PROGRAM UserMode
VAR

(*GapMode*)
	UserGapPositionNew:LREAL:=20;//target
	UserGapVelocityNew:LREAL:=1;//target
	UserGapPositionDisplay:LREAL;//current
	UserGapVelocityDisplay:LREAL;//current
	//
	(**)
	btn_UserGapMove:BOOL;
	btn_UserGapStop:BOOL;
	(*Var*)
	fb_ton1:TON;
	fb_ton2:TON;
	fb_ton3:TON;
	(*Status*)
	State:DINT;
	Busy:BOOL;
	InitPowerDone:BOOL;
	InitCompensationDatasDone:BOOL;
	(*FB*)
	m_state: DINT;
	n_state: DINT;
	s_state: DINT;
	(*¼ì²âµ½ÏÞÎ»£¬»Ö¸´Move×´Ì¬*)
	FTrig_ReachLS: F_TRIG;
	FTrig_btn_GapMove: F_TRIG;
	GapOutRange: BOOL;
	(*PowerOff*)
	d_state: DINT;
	i: INT;
	j: INT;
	k: INT;
	moni_State:DINT;
	TargetPosLessThanCurrentPos:BOOL;
	PositiveMoving:BOOL;
	HysteresisMoving:BOOL;
	NoneHysteresisMoving:BOOL;
	(*Spectroscopy scanning Mode*)
	IsSSMotionMode:BOOL;
	RegularMotionMode:BOOL;
	SSMotionMode:BOOL;
	SS_StepSize:LREAL:=0.001;
	SS_StepNumber:INT:=10;
	SS_StepVelocity:LREAL:=1;
	SS_Move:BOOL;
	SS_Stop:BOOL;
	SS_MoveState:DINT;
	SS_StopState:DINT;
	SS_currentStep:DINT:=0;
	SS_StepSystemTime_Begin:ARRAY[0..100] OF ULINT;
	SS_StepSystemTime_End:ARRAY[0..100] OF ULINT;
	SS_StepCountTime:ARRAY[0..100] OF ULINT;
	SS_TimeCountBegin:BOOL;
	m: INT;
	SS_TON: TON;
	StepEachTime:TIME;
	StepEachTime_ms:INT:=1000;//ms
	SS_OTSTRUCT :OTSTRUCT ;
	SS_StartPositionDisplay:LREAL;
	RTRG_SS_StartPositionDisplay:R_TRIG;
	SS_InitStartPositionDone:BOOL;
	
	//
	min_SS_StepSize	: LREAL:=0;
	max_SS_StepSize	: LREAL:=200;
	inRange_SS_StepSize	: BOOL;
	//
	min_SS_StepNumber	: INT:=1;
	max_SS_StepNumber	: INT:=1000;
	inRange_SS_StepNumber	: BOOL;
	//
	min_SS_StepVelocity:LREAL:=0;
	max_SS_StepVelocity:LREAL:=1;
	inRange_SS_StepVelocity:BOOL;
	//
	min_StepEachTime_ms:INT:=100;
	max_StepEachTime_ms:INT:=10000;
	inRange_StepEachTime_ms:BOOL;
	l: INT;
	testa: BOOL;
	testb: BOOL;
	Threshold_GapChangeFlag: LREAL;
	Threshold_TaperChangeFlag: LREAL;
	TaperAndGapSafetyfactor: LREAL:=1;
	
		//
	//Global Chain protection-MPS
	Global_ChainProtection_MPS_StorageRingReady:BOOL;
	Global_ChainProtection_MPS_On: BOOL;
	Global_ChainProtection_MPS_MaxGapValue: LREAL;
	Global_ChainProtection_MPS_MoveVelocity: LREAL;
	Global_ChainProtection_MPS_Done: BOOL;
	//Global_ChainProtection_Error: BOOL;
	//Global_ChainProtection_ErrorID: INT;
	//Global_ChainProtection_ErrorDescription: STRING;
	Global_ChainProtection_MPS_ManualOperation:BOOL:=TRUE;
	Global_ChainProtection_MPS_FTRIG:F_TRIG;
	Global_ChainProtection_MPS_FTRIG_Manul:F_TRIG;
	Global_ChainProtection_MPS_TON:TON;
	Global_ChainProtection_MPS_Triggered:BOOL;
	Global_ChainProtection_MPS_In:BOOL;
	Global_ChainProtection_MPS_In1 AT%I* :BOOL;//下降沿表示触发
	Global_ChainProtection_MPS_In2 AT%I* :BOOL;
	Global_ChainProtection_MPS_State:DINT;
	Global_ChainProtection_MPS_Out1 AT%Q* :BOOL;//上升沿标识到达最大间隙，连锁保护成功
	Global_ChainProtection_MPS_Out2 AT%Q* :BOOL;
	Global_ChainProtection_MPS_TON_Stop2Move:TON;
	Global_ChainProtection_MPS_TON_Stop2Move_InTaperMode:TON;
	Global_ChainProtection_MPS_TON_Power2Move:TON;
	//Global Chain protection-EPS
	Global_ChainProtection_EPS_BeamLineReady:BOOL;
	Global_ChainProtection_EPS_On: BOOL;
	Global_ChainProtection_EPS_MaxGapValue: LREAL;
	Global_ChainProtection_EPS_MoveVelocity: LREAL;
	Global_ChainProtection_EPS_Done: BOOL;
	//Global_ChainProtection_Error: BOOL;
	//Global_ChainProtection_ErrorID: INT;
	//Global_ChainProtection_ErrorDescription: STRING;
	Global_ChainProtection_EPS_ManualOperation:BOOL:=TRUE;
	Global_ChainProtection_EPS_FTRIG:F_TRIG;
	Global_ChainProtection_EPS_FTRIG_Manul:F_TRIG;
	Global_ChainProtection_EPS_TON:TON;
	Global_ChainProtection_EPS_Triggered:BOOL;
	Global_ChainProtection_EPS_In:BOOL;
	Global_ChainProtection_EPS_In1 AT%I* :BOOL;//下降沿表示触发
	Global_ChainProtection_EPS_In2 AT%I* :BOOL;
	Global_ChainProtection_EPS_State:DINT;
	Global_ChainProtection_EPS_Out1 AT%Q* :BOOL;//上升沿标识到达最大间隙，连锁保护成功
	Global_ChainProtection_EPS_Out2 AT%Q* :BOOL;
	Global_ChainProtection_EPS_TON_Stop2Move:TON;
	Global_ChainProtection_EPS_TON_Stop2Move_InTaperMode:TON;
	Global_ChainProtection_EPS_TON_Power2Move:TON;
	//
	Threshold_motorsTargetPosCalculate:LREAL;
	
	PhaseShifterLinPositionNewTemp: LREAL;
		//OneKeyToMaxGap
	btn_OneKeyToMaxGap:BOOL;
	OneKeyToMaxGap_RTRIG:R_TRIG;
	OneKeyToMaxGap_TON:TON;
	OneKeyToMaxGap_Triggered:BOOL;
	OneKeyToMaxGap_State:DINT;
	OneKeyToMaxGap_TON_Stop2Move:TON;
	OneKeyToMaxGap_TON_Stop2Move_InTaperMode:TON;
	OneKeyToMaxGap_TON_Power2Move:TON;
	OneKeyToMaxGap_Done:BOOL;
END_VAR

IF NOT PositionBiasDone THEN
	RETURN;
END_IF
IF NOT loadParametersDone THEN
	RETURN;
END_IF
(*btn_Power On/Off*)
IF btn_Power AND NOT st_Power THEN
	btn_PowerOn:=TRUE;
	btn_Power:=FALSE;
END_IF
IF btn_Power AND st_Power THEN
	btn_PowerOff:=TRUE;
	btn_Power:=FALSE;
END_IF
IF btn_PowerOn THEN
	A_PowerOn();
END_IF
IF btn_PowerOff THEN
	A_PowerOff();
END_IF


(*补偿数据处理*)
A_InitCompensationData();

(*常规磁间隙开合*)
IF RegularMotionMode AND NOT SSMotionMode THEN
	A_RegularMotion();
END_IF

(*Spectroscopy scanning Mode*)
IF IsSSMotionMode THEN
	SSMotionMode:=TRUE;
	RegularMotionMode:=FALSE;
ELSE
	SSMotionMode:=FALSE;
	RegularMotionMode:=TRUE;
END_IF
IF	SSMotionMode AND NOT RegularMotionMode THEN
	A_SpectroscopyScanningMotion();
END_IF

A_CheckMotorsPos();

(*GlobalChainProtection*)
A_GlobalChainProtection_MPS();
A_GlobalChainProtection_EPS();

(*A_OneKeyToMaxGap*)
A_OneKeyToMaxGap();

ACTION A_CheckMotorsPos:
//
//目标位置速度超出阈值判断
//
//gap posiion
IF UserGapPositionNew<min_UserGapPositionNew OR UserGapPositionNew>max_UserGapPositionNew THEN
	inRange_UserGapPositionNew:=FALSE;
END_IF
IF UserGapPositionNew>=min_UserGapPositionNew AND UserGapPositionNew<=max_UserGapPositionNew THEN
	inRange_UserGapPositionNew:=TRUE;
END_IF
//gap velocity
IF UserGapVelocityNew<min_UserGapVelocityNew OR UserGapVelocityNew>max_UserGapVelocityNew THEN
	inRange_UserGapVelocityNew:=FALSE;
END_IF
IF UserGapVelocityNew>=min_UserGapVelocityNew AND UserGapVelocityNew<=max_UserGapVelocityNew THEN
	inRange_UserGapVelocityNew:=TRUE;
END_IF
//SS Mode
IF SS_StepSize<min_SS_StepSize OR SS_StepSize>max_SS_StepSize THEN
	inRange_SS_StepSize:=FALSE;
END_IF
IF SS_StepSize>=min_SS_StepSize AND SS_StepSize<=max_SS_StepSize THEN
	inRange_SS_StepSize:=TRUE;
END_IF
IF SS_StepNumber<min_SS_StepNumber OR SS_StepNumber>max_SS_StepNumber THEN
	inRange_SS_StepNumber:=FALSE;
END_IF
IF SS_StepNumber>=min_SS_StepNumber AND SS_StepNumber<=max_SS_StepNumber THEN
	inRange_SS_StepNumber:=TRUE;
END_IF
IF SS_StepVelocity<min_SS_StepVelocity OR SS_StepVelocity>max_SS_StepVelocity THEN
	inRange_SS_StepVelocity:=FALSE;
END_IF
IF SS_StepVelocity>=min_SS_StepVelocity AND SS_StepVelocity<=max_SS_StepVelocity THEN
	inRange_SS_StepVelocity:=TRUE;
END_IF
IF StepEachTime_ms<min_StepEachTime_ms OR StepEachTime_ms>max_StepEachTime_ms THEN
	inRange_StepEachTime_ms:=FALSE;
END_IF
IF StepEachTime_ms>=min_StepEachTime_ms AND StepEachTime_ms<=max_StepEachTime_ms THEN
	inRange_StepEachTime_ms:=TRUE;
END_IF


//
//输入速度和位置保护
//
IF btn_UserGapMove  AND NOT SSMotionMode AND RegularMotionMode THEN
	IF NOT inRange_UserGapPositionNew THEN
		btn_UserGapStop:=TRUE;
		btn_UserGapMove:=FALSE;
		Error:=TRUE;
		ErrorId:=801;
		ErrorDescription:='target Gap position out of range,please check';
		RETURN;
	ELSE
		//btn_UserGapStop:=FALSE;
		Error:=FALSE;
		ErrorId:=0;
		ErrorDescription:='';	
	END_IF
	IF NOT inRange_UserGapVelocityNew THEN
		btn_UserGapStop:=TRUE;
		btn_UserGapMove:=FALSE;
		Error:=TRUE;
		ErrorId:=802;
		ErrorDescription:='target Gap velocity out of range,please check';
		RETURN;
	ELSE
		//btn_UserGapStop:=FALSE;
		Error:=FALSE;
		ErrorId:=0;
		ErrorDescription:='';
	END_IF
END_IF

//
//运动过程中，监控目标位置速度
//
IF moveStatusPhaseShifterLin THEN
	IF NOT inRange_UserGapPositionNew THEN
		btn_UserGapStop:=TRUE;
		Error:=TRUE;
		ErrorId:=805;
		ErrorDescription:='target Gap position out of range in moving process!';
		FB_PlcEmergencyStop();
	END_IF
	IF NOT inRange_UserGapVelocityNew THEN
		btn_UserGapStop:=TRUE;
		Error:=TRUE;
		ErrorId:=806;
		ErrorDescription:='target Gap velocity out of range in moving process!';
		FB_PlcEmergencyStop();
	END_IF
END_IF
//
//运动过程中，监控每一个轴的目标位置，目标位置若超出阈值，Emergency
//
IF moveStatusPhaseShifterLin THEN
		IF PhaseShifterLinPositionNew<min_UserGapPositionNew OR PhaseShifterLinPositionNew>max_UserGapPositionNew THEN
			btn_UserGapStop:=TRUE;
			Error:=TRUE;
			ErrorId:=809;
			ErrorDescription:='target PhaseShifterLinPositionNew out of range in moving process!';
			FB_PlcEmergencyStop();
		END_IF
END_IF
END_ACTION

ACTION A_GlobalChainProtection_EPS:
//硬线输入定义
Global_ChainProtection_EPS_In:=Global_ChainProtection_EPS_In1 AND Global_ChainProtection_EPS_In2;
//硬线输出定义
Global_ChainProtection_EPS_Out1:=Global_ChainProtection_EPS_Done;
Global_ChainProtection_EPS_Out2:=Global_ChainProtection_EPS_Done;
//总开关
IF NOT Global_ChainProtection_EPS_On THEN
	RETURN;
END_IF
//判断插入件状态，是否就位
//IF NOT IDControlReady THEN
//	Global_ChainProtection_EPS_Done:=FALSE;
//	Error:= TRUE;
//	ErrorID:= 1501;
//	ErrorDescription:='ID NOT READY!';
//	RETURN;
//END_IF
//判断储存环是否给出就位信号，暂时由参数表给出TRUE，最终将由IOC接受PV
IF 	NOT Global_ChainProtection_EPS_BeamLineReady THEN
	Global_ChainProtection_EPS_Done:=FALSE;
	Error:= TRUE;
	ErrorID:= 1503;
	ErrorDescription:='Global_ChainProtection_EPS_BeamLineReady NOT Ready';
	RETURN;
END_IF
//
//全局连锁保护程序开始
//
//0.检测到下降沿，触发
//1.判断电机是否在开启状态,没有就打开电源
//2.判断是否在Moving状态,若有就Stop
//3.将磁间隙打开到至最大阈值
//4.到位后给出反馈，且安全PLC触发
Global_ChainProtection_EPS_FTRIG(CLK:=Global_ChainProtection_EPS_In);
IF Global_ChainProtection_EPS_FTRIG.Q THEN
	Global_ChainProtection_EPS_Triggered:=TRUE;
END_IF
Global_ChainProtection_EPS_FTRIG_Manul(CLK:=Global_ChainProtection_EPS_ManualOperation);
IF Global_ChainProtection_EPS_FTRIG_Manul.Q THEN
	Global_ChainProtection_EPS_Triggered:=TRUE;
END_IF
IF Global_ChainProtection_EPS_Triggered THEN
	CASE Global_ChainProtection_EPS_State OF
		0://1.判断电机是否在开启状态,没有就打开电源
			IF st_Power=1 THEN
				Global_ChainProtection_EPS_State:=1;
			ELSE
				btn_PowerOn:=TRUE;
				IF btn_PowerOn THEN
					A_PowerOn();
				END_IF
			END_IF
		1://1.判断是否在谱学扫描模式，如果是，则切换回正常运动模式
			IF IsSSMotionMode THEN
				SS_Stop:=TRUE;
				IsSSMotionMode:=FALSE;
			END_IF
			Global_ChainProtection_EPS_State:=2;
		2://判断是否在taper，如果在taper,则判断是否在运动，如果是，则停止运动,0.5sh后，转入下一步
			(*IF TaperOrNot THEN
				IF moveStatusLeftTop OR moveStatusRightTop OR moveStatusLeftBottom OR moveStatusRightBottom THEN
					btn_UserGapStop:=TRUE;
				ELSE
					Global_ChainProtection_EPS_TON_Stop2Move_InTaperMode(PT:=T#0.5S);
					Global_ChainProtection_EPS_TON_Stop2Move_InTaperMode.IN:=TRUE;
					IF Global_ChainProtection_EPS_TON_Stop2Move_InTaperMode.Q THEN
						TaperOrNot:=FALSE;//关闭taper模式
						Global_ChainProtection_EPS_State:=3;
					END_IF
				END_IF
			ELSE
			*)
				Global_ChainProtection_EPS_State:=3;
			//END_IF
		3://3.判断是否在Moving状态,若有就Stop.Taper模式已处理完，此处开始走正常GAP开合逻辑
			IF moveStatusPhaseShifterLin THEN
				btn_UserGapStop:=TRUE;
			ELSE
				Global_ChainProtection_EPS_TON_Stop2Move(PT:=T#0.5S);
				Global_ChainProtection_EPS_TON_Stop2Move.IN:=TRUE;
				IF Global_ChainProtection_EPS_TON_Stop2Move.Q THEN
					Global_ChainProtection_EPS_State:=4;
				END_IF
			END_IF
		4://当前磁间隙如何和最大磁间隙差别不大，不超过0.1，则直接保护
			IF ABS(UserGapPositionDisplay-Global_ChainProtection_EPS_MaxGapValue)<=0.1 THEN
				Global_ChainProtection_EPS_Done:=TRUE;
				Plc_EmergencyStop:=FALSE;	
				Error:=TRUE;
				ErrorID:=1506;
				ErrorDescription:='EPS Triggered,but ABS(UserGapPositionDisplay-Global_ChainProtection_EPS_MaxGapValue)<=0.1 ';	
			ELSE
				Global_ChainProtection_EPS_State:=5;
			END_IF
		5://5.将磁间隙打开到至最大阈值
			Global_ChainProtection_EPS_TON(PT:=INT_TO_TIME(LREAL_TO_INT(Global_ChainProtection_EPS_MaxGapValue/Global_ChainProtection_EPS_MoveVelocity+30))*1000);
			Global_ChainProtection_EPS_TON.IN:=TRUE;
			Global_ChainProtection_EPS_TON_Power2Move(PT:=T#0.1S);
			Global_ChainProtection_EPS_TON_Power2Move.IN:=TRUE;
			UserGapPositionNew:=Global_ChainProtection_EPS_MaxGapValue;
			UserGapVelocityNew:=Global_ChainProtection_EPS_MoveVelocity;
			btn_UserGapMove:=TRUE;
			IF Global_ChainProtection_EPS_TON_Power2Move.Q THEN
				IF FB_MOVE.BCGapDone THEN
					Global_ChainProtection_EPS_State:=88;
				END_IF
			END_IF
			IF Global_ChainProtection_EPS_TON.Q THEN//如果150s后，还没有运动到指定gap，则报错
				Global_ChainProtection_EPS_State:=-100;
			END_IF
		88://4.到位后给出反馈，且安全PLC触发
			Global_ChainProtection_EPS_Done:=TRUE;
			Plc_EmergencyStop:=FALSE;	
			Error:=TRUE;
			ErrorID:=1504;
			ErrorDescription:='Global_ChainProtection_EPS Triggered ';	
		-100:
			Global_ChainProtection_EPS_Done:=FALSE;
			Error:=TRUE;
			ErrorID:=1505;
			ErrorDescription:='NOT MOVING TO MAXGAP';
	END_CASE
END_IF
END_ACTION

ACTION A_GlobalChainProtection_MPS:
//硬线输入定义
Global_ChainProtection_MPS_In:=Global_ChainProtection_MPS_In1 AND Global_ChainProtection_MPS_In2;
//硬线输出定义
Global_ChainProtection_MPS_Out1:=Global_ChainProtection_MPS_Done;
Global_ChainProtection_MPS_Out2:=Global_ChainProtection_MPS_Done;
//总开关
IF NOT Global_ChainProtection_MPS_On THEN
	RETURN;
END_IF
//判断插入件状态，是否就位
//IF NOT IDControlReady THEN
//	Global_ChainProtection_MPS_Done:=FALSE;
//	Error:= TRUE;
//	ErrorID:= 1401;
//	ErrorDescription:='ID NOT READY!';
//	RETURN;
//END_IF
//判断储存环是否给出就位信号，暂时由参数表给出TRUE，最终将由IOC接受PV
IF 	NOT Global_ChainProtection_MPS_StorageRingReady THEN
	Global_ChainProtection_MPS_Done:=FALSE;
	Error:= TRUE;
	ErrorID:= 1403;
	ErrorDescription:='StorageRingChainProtection NOT Ready';
	RETURN;
END_IF
//
//全局连锁保护程序开始
//
//0.检测到下降沿，触发
//1.判断电机是否在开启状态,没有就打开电源
//2.判断是否在Moving状态,若有就Stop
//3.将磁间隙打开到至最大阈值
//4.到位后给出反馈，且安全PLC触发
Global_ChainProtection_MPS_FTRIG(CLK:=Global_ChainProtection_MPS_In);
IF Global_ChainProtection_MPS_FTRIG.Q THEN
	Global_ChainProtection_MPS_Triggered:=TRUE;
END_IF
Global_ChainProtection_MPS_FTRIG_Manul(CLK:=Global_ChainProtection_MPS_ManualOperation);
IF Global_ChainProtection_MPS_FTRIG_Manul.Q THEN
	Global_ChainProtection_MPS_Triggered:=TRUE;
END_IF
IF Global_ChainProtection_MPS_Triggered THEN
	CASE Global_ChainProtection_MPS_State OF
		0://1.判断电机是否在开启状态,没有就打开电源
			IF st_Power=1 THEN
				Global_ChainProtection_MPS_State:=1;
			ELSE
				btn_PowerOn:=TRUE;
				IF btn_PowerOn THEN
					A_PowerOn();
				END_IF
			END_IF
		1://1.判断是否在谱学扫描模式，如果是，则切换回正常运动模式
			IF IsSSMotionMode THEN
				SS_Stop:=TRUE;
				IsSSMotionMode:=FALSE;
			END_IF
			Global_ChainProtection_MPS_State:=2;
		2://判断是否在taper，如果在taper,则判断是否在运动，如果是，则停止运动,0.5sh后，转入下一步
			(*IF TaperOrNot THEN
				IF moveStatusLeftTop OR moveStatusRightTop OR moveStatusLeftBottom OR moveStatusRightBottom THEN
					btn_UserGapStop:=TRUE;
				ELSE
					Global_ChainProtection_MPS_TON_Stop2Move_InTaperMode(PT:=T#0.5S);
					Global_ChainProtection_MPS_TON_Stop2Move_InTaperMode.IN:=TRUE;
					IF Global_ChainProtection_MPS_TON_Stop2Move_InTaperMode.Q THEN
						TaperOrNot:=FALSE;//关闭taper模式
						Global_ChainProtection_MPS_State:=3;
					END_IF
				END_IF
			ELSE
			*)
				Global_ChainProtection_MPS_State:=3;
			//END_IF
		3://3.判断是否在Moving状态,若有就Stop.Taper模式已处理完，此处开始走正常GAP开合逻辑
			IF moveStatusPhaseShifterLin THEN
				btn_UserGapStop:=TRUE;
			ELSE
				Global_ChainProtection_MPS_TON_Stop2Move(PT:=T#0.5S);
				Global_ChainProtection_MPS_TON_Stop2Move.IN:=TRUE;
				IF Global_ChainProtection_MPS_TON_Stop2Move.Q THEN
					Global_ChainProtection_MPS_State:=4;
				END_IF
			END_IF
		4://当前磁间隙如何和最大磁间隙差别不大，不超过0.1，则直接保护
			IF ABS(UserGapPositionDisplay-Global_ChainProtection_MPS_MaxGapValue)<=0.1 THEN
				Global_ChainProtection_MPS_Done:=TRUE;
				Plc_EmergencyStop:=FALSE;	
				Error:=TRUE;
				ErrorID:=1406;
				ErrorDescription:='MPS Triggered,but ABS(UserGapPositionDisplay-Global_ChainProtection_MPS_MaxGapValue)<=0.1 ';	
			ELSE
				Global_ChainProtection_MPS_State:=5;
			END_IF
		5://5.将磁间隙打开到至最大阈值
			Global_ChainProtection_MPS_TON(PT:=INT_TO_TIME(LREAL_TO_INT(Global_ChainProtection_MPS_MaxGapValue/Global_ChainProtection_MPS_MoveVelocity+30))*1000);
			Global_ChainProtection_MPS_TON.IN:=TRUE;
			Global_ChainProtection_MPS_TON_Power2Move(PT:=T#0.1S);
			Global_ChainProtection_MPS_TON_Power2Move.IN:=TRUE;
			UserGapPositionNew:=Global_ChainProtection_MPS_MaxGapValue;
			UserGapVelocityNew:=Global_ChainProtection_MPS_MoveVelocity;
			btn_UserGapMove:=TRUE;
			IF Global_ChainProtection_MPS_TON_Power2Move.Q THEN
				IF FB_MOVE.BCGapDone THEN
					Global_ChainProtection_MPS_State:=88;
				END_IF
			END_IF
			IF Global_ChainProtection_MPS_TON.Q THEN//如果150s后，还没有运动到指定gap，则报错
				Global_ChainProtection_MPS_State:=-100;
			END_IF
		88://4.到位后给出反馈，且安全PLC触发
			Global_ChainProtection_MPS_Done:=TRUE;
			Plc_EmergencyStop:=FALSE;	
			Error:=TRUE;
			ErrorID:=1404;
			ErrorDescription:='Global_ChainProtection_MPS Triggered ';	
		-100:
			Global_ChainProtection_MPS_Done:=FALSE;
			Error:=TRUE;
			ErrorID:=1405;
			ErrorDescription:='NOT MOVING TO MAXGAP';
	END_CASE
END_IF
END_ACTION

ACTION A_InitCompensationData:
(*补偿开始*)
IF USE_SingleAxis_Compensation THEN
	//
	//1.目标位置解算
	//
	//左轴目标位置解算
	FOR	i:= 1 TO 17 DO
			IF UserGapPositionNew<M_Compensation[i+1].Gap AND UserGapPositionNew>=M_Compensation[i].Gap THEN
				IF i<>18 THEN
					PhaseShifterLinPositionNew:=(((UserGapPositionNew-M_Compensation[i].Gap)*(M_Compensation[i+1].PhaseShifterLin-M_Compensation[i].PhaseShifterLin))
							/(M_Compensation[i+1].Gap-M_Compensation[i].Gap))+M_Compensation[i].PhaseShifterLin;
					M_CompensationNumber:=i;
					InitCompensationDatasDone:=TRUE;
				ELSIF i=18 AND UserGapPositionNew=M_Compensation[i].Gap THEN		(*Gap=14µÄÌØÊâÇé¿ö*)
					(**)
					PhaseShifterLinPositionNew:=M_Compensation[i].PhaseShifterLin;
					M_CompensationNumber:=i;
					InitCompensationDatasDone:=TRUE;
				ELSE
					PhaseShifterLinPositionNew:=UserGapPositionNew;
					M_CompensationNumber:=i;
					InitCompensationDatasDone:=TRUE;
				END_IF
			END_IF
	END_FOR

	//显示位置反解算
	FOR k:= 1 TO 17 DO
			IF Pos_PhaseShifterLin<M_Compensation[k+1].PhaseShifterLin AND Pos_PhaseShifterLin>=M_Compensation[k].PhaseShifterLin THEN
				UserGapPositionDisplay:=((Pos_PhaseShifterLin-M_Compensation[k].PhaseShifterLin)*(M_Compensation[k+1].Gap-M_Compensation[k].Gap))
											/(M_Compensation[k+1].PhaseShifterLin-M_Compensation[k].PhaseShifterLin)+M_Compensation[k].Gap;
				UserGapPositionDisplay:=DINT_TO_LREAL(LREAL_TO_DINT(UserGapPositionDisplay*100000))/100000;
			END_IF
	END_FOR
END_IF
(*速度可以不用解算，直接用即可*)
PhaseShifterLinVelocityDisplay:=Velo_PhaseShifterLin;
//Gap velocity
UserGapVelocityDisplay:=DINT_TO_LREAL(LREAL_TO_DINT(PhaseShifterLinVelocityDisplay*100000))/100000;


(*解算单轴位置后，核验并做保护*)
IF ABS(PhaseShifterLinPositionNew-UserGapPositionNew)>Threshold_motorsTargetPosCalculate THEN
	ErrorID:=1601;
	Error:=TRUE;
	ErrorDescription:='Threshold_motorsTargetPosCalculate';
	FB_PlcEmergencyStop();
END_IF
END_ACTION

ACTION A_OneKeyToMaxGap:
//0.上升沿触发
//1.判断电机是否在开启状态,没有就打开电源
//2.判断是否在Moving状态,若有就Stop
//3.将磁间隙打开到至最大阈值
//4.到位后给出反馈
OneKeyToMaxGap_RTRIG(CLK:=btn_OneKeyToMaxGap);
IF OneKeyToMaxGap_RTRIG.Q THEN
	OneKeyToMaxGap_Triggered:=TRUE;
	OneKeyToMaxGap_Done:=FALSE;
END_IF
IF OneKeyToMaxGap_Triggered THEN
	CASE OneKeyToMaxGap_State OF
		0://1.判断电机是否在开启状态,没有就打开电源
			IF st_Power=1 THEN
				OneKeyToMaxGap_State:=1;
			ELSE
				btn_PowerOn:=TRUE;
				IF btn_PowerOn THEN
					A_PowerOn();
				END_IF
			END_IF
		1://1.判断是否在谱学扫描模式，如果是，则切换回正常运动模式
			IF IsSSMotionMode THEN
				SS_Stop:=TRUE;
				IsSSMotionMode:=FALSE;
			END_IF
			OneKeyToMaxGap_State:=2;
		2://判断是否在taper，如果在taper,则判断是否在运动，如果是，则停止运动,0.5sh后，转入下一步
			//IF TaperOrNot THEN
			//	IF moveStatusLeftTop OR moveStatusRightTop OR moveStatusLeftBottom OR moveStatusRightBottom THEN
			//		btn_UserGapStop:=TRUE;
			//	ELSE
			//		OneKeyToMaxGap_TON_Stop2Move_InTaperMode(PT:=T#0.5S);
			//		OneKeyToMaxGap_TON_Stop2Move_InTaperMode.IN:=TRUE;
			//		IF OneKeyToMaxGap_TON_Stop2Move_InTaperMode.Q THEN
			//			TaperOrNot:=FALSE;//关闭taper模式
			//			OneKeyToMaxGap_State:=3;
			//			OneKeyToMaxGap_TON_Stop2Move_InTaperMode.IN:=FALSE;
			//		END_IF
			//	END_IF
			//ELSE
				OneKeyToMaxGap_State:=3;
			//END_IF
		3://3.判断是否在Moving状态,若有就Stop.Taper模式已处理完，此处开始走正常GAP开合逻辑
			IF moveStatusPhaseShifterLin THEN
				btn_UserGapStop:=TRUE;
			ELSE
				OneKeyToMaxGap_TON_Stop2Move(PT:=T#0.5S);
				OneKeyToMaxGap_TON_Stop2Move.IN:=TRUE;
				IF OneKeyToMaxGap_TON_Stop2Move.Q THEN
					OneKeyToMaxGap_State:=4;
					OneKeyToMaxGap_TON_Stop2Move.IN:=FALSE;
				END_IF
			END_IF
		4://4.将磁间隙打开到至最大阈值
			OneKeyToMaxGap_TON(PT:=INT_TO_TIME(LREAL_TO_INT(max_UserGapPositionNew+30))*1000);
			OneKeyToMaxGap_TON.IN:=TRUE;
			OneKeyToMaxGap_TON_Power2Move(PT:=T#0.1S);
			OneKeyToMaxGap_TON_Power2Move.IN:=TRUE;
			UserGapPositionNew:=max_UserGapPositionNew;
			UserGapVelocityNew:=1;
			btn_UserGapMove:=TRUE;
			IF OneKeyToMaxGap_TON_Power2Move.Q THEN
				OneKeyToMaxGap_TON_Power2Move.IN:=FALSE;
				IF FB_MOVE.BCGapDone THEN
					OneKeyToMaxGap_State:=88;
				END_IF
			END_IF
			IF OneKeyToMaxGap_TON.Q THEN//如果150s后，还没有运动到指定gap，则报错
				OneKeyToMaxGap_TON.IN:=FALSE;
				OneKeyToMaxGap_State:=-100;
			END_IF
			IF  btn_UserGapStop THEN
				//
				OneKeyToMaxGap_State:=0;
				OneKeyToMaxGap_Triggered:=FALSE;
				btn_OneKeyToMaxGap:=FALSE;
				OneKeyToMaxGap_Triggered:=FALSE;
				OneKeyToMaxGap_State:=0;
			END_IF
		88://6.到位后给出反馈
			OneKeyToMaxGap_Done:=TRUE;	
			Error:=FALSE;
			ErrorID:=0;
			ErrorDescription:='';
			btn_OneKeyToMaxGap:=FALSE;
			OneKeyToMaxGap_Triggered:=FALSE;
			OneKeyToMaxGap_State:=0;
				
		-100:
			OneKeyToMaxGap_Done:=FALSE;
			Error:=TRUE;
			ErrorID:=1705;
			ErrorDescription:='OneKeyToMaxGap Fail';
			btn_OneKeyToMaxGap:=FALSE;
			OneKeyToMaxGap_Triggered:=FALSE;
			OneKeyToMaxGap_State:=0;
	END_CASE
END_IF
END_ACTION

ACTION A_PowerOff:
CASE d_state OF
		0:(*PowerOff*)
			FB_Power(Off:=TRUE);
				d_state:=1;
		1:
			IF NOT FB_power.OffStatus THEN
				d_state:=1;
			ELSE
				d_state:=88;
			END_IF
		88:(*ResetAllState*)
			btn_PowerOn:=FALSE;
			btn_UserGapMove:=FALSE;
			btn_UserGapStop:=FALSE;
			fb_ton1.IN:=FALSE;
			fb_ton2.IN:=FALSE;
			fb_ton3.IN:=FALSE;
			State:=0;
			Busy:=FALSE;
			InitPowerDone:=FALSE;
			InitCompensationDatasDone:=FALSE;
			Error:=FALSE;
			ErrorID:=0;
			m_state:=0;
			n_state:=0;
			s_state:=0;
			btn_PowerOff:=FALSE;
			d_state:=0;
			Led_Run:=FALSE;
			Led_Error:=FALSE;
			moni_State:=0;
			i:=0;
END_CASE
END_ACTION

ACTION A_PowerOn:
(****************************************************************
NAME:			A_PowerOn
DATA:			2018.1.9
VERSION:		1.0.0
DESCRIPTION:	
				ÉÏµãÃüÁîºó£¬Ë³ÐòÖ´ÐÐ£º
				1.FB_PowerOn
				·µ»ØÖ´ÐÐÊÇ·ñ³É¹¦
HISTORY:
				2019.1.9		NEW

***************************************************************)
fb_ton3(PT:=t#0.5s);
CASE State OF
	0:	(*FB_Power_On*)
		FB_Power(On:=TRUE);
		fb_ton3.IN:=TRUE;
		State:=1;
	1:	(*wait*)
		FB_power();
		IF NOT FB_power.OnStatus THEN		(*FB_Power_OnÃ»ÓÐÖ´ÐÐÍê£¬wait£¬³¬Ê±FB Error*)
			IF NOT fb_ton3.Q THEN
				State:=1;
			ELSE
				ErrorID:=1;
				State:=99;
			END_IF
		ELSE
			State:=88;
		END_IF
	88:	(*All Done*)
		btn_PowerOn:=FALSE;
		State:=0;
		Error:=FALSE;
		ErrorID:=0;
		Busy:=FALSE;
		InitPowerDone:=TRUE;
		FB_power.On:=FALSE;
		fb_ton3.IN:=FALSE;
		LED_Error:=FALSE;
	99:
		Error:=TRUE;
		//ErrorID:=701;
		//ErrorDescription:='power on error';		
		btn_PowerOn:=FALSE;
		State:=99;
		Busy:=FALSE;
		InitPowerDone:=FALSE;
		fb_ton3.IN:=FALSE;
		LED_Error:=TRUE;
END_CASE
END_ACTION

ACTION A_RegularMotion:

(*分别比较四轴目标位置与当前位置的差，如果目标位置比当前位置低，则需要运动到更低-回程差一半；再运动至最终目标位置*)
//只在m=和n=0的时候判断，否则会出现一些BUG，比如往大间隙开时，运动到位后m不能回到0.
IF m_state=0 AND n_state=0 THEN
		TargetPosLessThanCurrentPos:=FALSE;
	IF PhaseShifterLinPositionNew-Pos_PhaseShifterLin<-LEDriftErrorThreshold THEN
			TargetPosLessThanCurrentPos:=TRUE;
	END_IF
END_IF

(*Move*)
IF InitCompensationDatasDone THEN
		(*四轴目标位置都大于当前位置，直接走到目标位置即可，不需要先走到考虑回城误差的临时位置*)
		IF NOT TargetPosLessThanCurrentPos AND NOT HysteresisMoving THEN
			CASE m_state OF
				0:
					FB_Move.Mode:=1;						//1.gap;2.single;3.taper;4.debug;5.BCGap&UserMode		
					FB_Move.PowerState:=st_Power;						
			
					IF btn_UserGapMove THEN				
						moveStatusGap:=TRUE;
						FB_Move.BCGapReset:=TRUE;
						IF NOT st_Power THEN
							ErrorID:=1501;
							Error:=TRUE;
							ErrorDescription:='Plz PowerOn Frist';
							LED_Error:=TRUE;
							//btn_UserGapMove:=FALSE;
							RETURN;
						ELSE
							ErrorID:=0;
							Error:=FALSE;
							ErrorDescription:='';
							LED_Error:=FALSE;
							//btn_UserGapMove:=TRUE;
						END_IF
						//目标速度位置赋值
						FB_Move.TargetGapPosition:=PhaseShifterLinPositionNew;
						FB_Move.TargetGapVelocity:=UserGapVelocityNew;

						m_state:=1;
						FB_Move();
					END_IF
				1:						
					FB_Move.BCGapMove:=TRUE;
					btn_UserGapMove:=FALSE;
					FB_Move();
					IF NOT FB_Move.BCGapDone THEN	
						Led_Run:=TRUE;
						m_state:=1;
					ELSE				
						m_state:=88;
					END_IF
				88:
					moveStatusGap:=FALSE;
					btn_UserGapMove:=FALSE;		
					Led_Run:=FALSE;
					m_state:=0;
			END_CASE
		(*四轴有目标位置小于当前位置，先走到临时位置，再走到目标位置*)
		ELSE
			CASE n_state OF
				0:
					FB_Move.Mode:=1;						//1.gap;2.single;3.taper;4.debug;5.BCGap&UserMode;5:userMode_2		
					FB_Move.PowerState:=st_Power;			
					IF btn_UserGapMove THEN	
						FB_Move.BCGapReset:=TRUE;					
						moveStatusGap:=TRUE;
						IF NOT st_Power THEN
							ErrorID:=1501;
							Error:=TRUE;
							ErrorDescription:='Plz PowerOn Frist';
							LED_Error:=TRUE;
							//btn_UserGapMove:=FALSE;
							RETURN;
						ELSE
							ErrorID:=0;
							Error:=FALSE;
							ErrorDescription:='';
							LED_Error:=FALSE;
							//btn_UserGapMove:=TRUE;
						END_IF						
						//
						IF TargetPosLessThanCurrentPos THEN			
							FB_Move.TargetGapPosition:=PhaseShifterLinPositionNew-HysteresisError;
						ELSE
							FB_Move.TargetGapPosition:=PhaseShifterLinPositionNew;	
						END_IF
						//	
						//	close gap情况下，加入了LeftTopLinPositionNewTemp。//
						//如果在往小间隙运行过程中，改变了目标gap，会在第到达第一次目标位置后，继续向第二
						//次输入的目标运动，而不会回到第一次的目标位置。用temp锁定目标位置
						PhaseShifterLinPositionNewTemp:=PhaseShifterLinPositionNew;
						FB_Move.TargetGapVelocity:=UserGapVelocityNew;
						IF UserGapVelocityNew >1 THEN								  
							ErrorID:=1502;
							Error:=TRUE;
							ErrorDescription:='UserGapVelocityNew must<=1';
							LED_Error:=TRUE;
							btn_UserGapMove:=FALSE;
							RETURN;
						ELSE
							ErrorID:=0;
							Error:=FALSE;
							ErrorDescription:='';
							LED_Error:=FALSE;	
						END_IF										

						FB_Move();
						HysteresisMoving:=TRUE;		
						n_state:=1;	
					END_IF
				1:
					btn_UserGapMove:=FALSE;	
					FB_Move.BCGapMove:=TRUE;
					FB_Move();
					IF NOT FB_Move.BCGapDone THEN			(*还未运动到位置,运动过程中*)
						Led_Run:=TRUE;
						n_state:=1;
					ELSE									
						n_state:=2;							(*转到下一步，运动到最终位置*)
						FB_Move.BCGapMove:=FALSE;
						//Led_Run:=FALSE;
					END_IF
				2:
					FB_Move.BCGapReset:=FALSE;
					FB_Move.Mode:=1;						//1.gap;2.single;3.taper;4.debug;5.BCGap&UserMode		
					FB_Move.PowerState:=st_Power;			
					FB_Move.BCGapMove:=TRUE;
					//直接走到目标位置，已经走到位置的，可以继续下命令，只不过它不在走了而已
					FB_Move.TargetGapPosition:=PhaseShifterLinPositionNewTemp;
					FB_Move.TargetGapVelocity:=UserGapVelocityNew;

					FB_Move();							
					n_state:=3;
				3:
					FB_Move();
					IF NOT FB_Move.BCGapDone THEN			(*还未运动到位置,运动过程中*)
						Led_Run:=TRUE;
						n_state:=3;
					ELSE									
						n_state:=88;							(*运动到了最终位置*)
					END_IF
					(*
					IF NOT Unreach_LS_Bottom THEN
						n_state:=88;							(*在运动过程中如果碰到下限位，则也转到下一步，运动到最终位置*)
						FB_Move.BCGapMove_2:=FALSE;
					END_IF
					*)
				88:				
					moveStatusGap:=FALSE;
					btn_UserGapMove:=FALSE;				
					Led_Run:=FALSE;
					n_state:=0;
					HysteresisMoving:=FALSE;
			END_CASE
		END_IF
	//
	//FB_Move.BCLeftTopPosition等四轴位置监控
	//
END_IF


CASE s_state OF
	0:
		IF btn_UserGapStop OR btn_Reset THEN					
			moveStatusGap:=FALSE;
			m_state:=0;	
			n_state:=0;	
			HysteresisMoving:=FALSE;
			
			FB_Stop.Mode:=1;	
			FB_Stop.PowerState:=st_Power;
			FB_Stop.BCGapStop:=TRUE;
			FB_Stop();	
			s_state:=1;
		END_IF
	1:
		btn_UserGapStop:=FALSE;	
		FB_Stop();
		IF NOT FB_Stop.BCGapDone THEN
			s_state:=1;
		ELSE
			s_state:=88;
		END_IF
	88:
		FB_Move.BCGapReset:=FALSE;
		btn_reset:=FALSE;
		s_state:=0;
END_CASE


(*触发限位开关后，相当于点击了Stop按钮*)
FTrig_ReachLS(CLK:=Unreach_LS_Far AND Unreach_LS_Near);
IF FTrig_ReachLS.Q THEN
	btn_UserGapStop:=TRUE;
END_IF
(*触发限位后，如果继续向前运动，点击move，则相当于点击stop，用于恢复move的状态位*)
IF NOT Unreach_LS_Far AND btn_UserGapMove AND UserGapPositionNew >= UserGapPositionDisplay THEN
	btn_UserGapStop:=TRUE;
END_IF
IF NOT Unreach_LS_Near AND btn_UserGapMove AND UserGapPositionNew <= UserGapPositionDisplay THEN
	btn_UserGapStop:=TRUE;
END_IF
END_ACTION

ACTION A_SpectroscopyScanningMotion:
(*输入保护*)
IF SS_Move AND SSMotionMode AND NOT RegularMotionMode THEN
	IF NOT inRange_SS_StepSize THEN
		SS_Stop:=TRUE;
		SS_Move:=FALSE;
		Error:=TRUE;
		ErrorId:=805;
		ErrorDescription:='target StepSize out of range,please check';
		RETURN;
	ELSE
		//SS_Stop:=FALSE;
		Error:=FALSE;
		ErrorId:=0;
		ErrorDescription:='';	
	END_IF
	//
	IF NOT inRange_SS_StepNumber THEN
		SS_Stop:=TRUE;
		SS_Move:=FALSE;
		Error:=TRUE;
		ErrorId:=806;
		ErrorDescription:='target StepNumber out of range,please check';
		RETURN;
	ELSE
		//SS_Stop:=FALSE;
		Error:=FALSE;
		ErrorId:=0;
		ErrorDescription:='';	
	END_IF
	IF NOT inRange_SS_StepVelocity THEN
		SS_Stop:=TRUE;
		SS_Move:=FALSE;
		Error:=TRUE;
		ErrorId:=807;
		ErrorDescription:='target StepVelocity out of range,please check';
		RETURN;
	ELSE
		//SS_Stop:=FALSE;
		Error:=FALSE;
		ErrorId:=0;
		ErrorDescription:='';	
	END_IF
	IF NOT inRange_StepEachTime_ms THEN
		SS_Stop:=TRUE;
		SS_Move:=FALSE;
		Error:=TRUE;
		ErrorId:=808;
		ErrorDescription:='target StepEachTime_ms out of range,please check';
		RETURN;
	ELSE
		//SS_Stop:=FALSE;
		Error:=FALSE;
		ErrorId:=0;
		ErrorDescription:='';	
	END_IF
END_IF
(*单步时长转换*)
StepEachTime:=INT_TO_TIME(StepEachTime_ms);
SS_TON(PT:=StepEachTime);
(*上升沿触发，初始SS位置=当前磁间隙*)
RTRG_SS_StartPositionDisplay(CLK:=SS_Move);
IF RTRG_SS_StartPositionDisplay.Q THEN
	SS_StartPositionDisplay:=UserGapPositionDisplay;
	SS_InitStartPositionDone:=TRUE;
END_IF
(*SS主程序*)
IF InitPowerDone AND InitCompensationDatasDone AND SS_Move AND SS_InitStartPositionDone THEN
	CASE SS_MoveState OF
		0:
				//UserGapPositionNew:=UserGapPositionDisplay+SS_StepSize;
				UserGapPositionNew:=SS_StartPositionDisplay+SS_StepSize*(SS_currentStep+1);
				A_InitCompensationData();
				FB_Move.Mode:=1;						//1.gap;2.single;3.taper;4.debug;5.BCGap&UserMode		
				FB_Move.PowerState:=st_Power;							
				FB_Move.TargetGapPosition:=PhaseShifterLinPositionNew;
				FB_Move.TargetGapVelocity:=UserGapVelocityNew;		
				FB_Move.BCGapMove:=TRUE;
				FB_Move();
				SS_MoveState:=1;
		1:
				SS_TON.IN:=TRUE;
				FB_Move();
				IF FB_Move.GapMoving AND NOT SS_TimeCountBegin THEN
					SS_StepSystemTime_Begin[SS_currentStep]:=F_GetSysTime();
					SS_TimeCountBegin:=TRUE;
				END_IF
				IF NOT FB_Move.BCGapDone THEN			
					Led_Run:=TRUE;
					SS_MoveState:=1;
				ELSE									
					SS_MoveState:=66;
					SS_StepSystemTime_End[SS_currentStep]:=F_GetSysTime();
					SS_StepCountTime[SS_currentStep]:=SS_StepSystemTime_End[SS_currentStep]-SS_StepSystemTime_Begin[SS_currentStep];
					SS_TimeCountBegin:=FALSE;
				END_IF
		66:
				SS_currentStep:=SS_currentStep+1;			
				Led_Run:=FALSE;
				IF SS_currentStep=SS_StepNumber THEN								
					SS_MoveState:=88;
				END_IF
				IF SS_currentStep<SS_StepNumber THEN
					SS_MoveState:=77;
				END_IF
		77://等待单步时长够
				IF SS_TON.Q THEN
					SS_TON.IN:=FALSE;
					SS_MoveState:=0;
				END_IF
		88:
				SS_TON.IN:=FALSE;
				SS_Move:=FALSE;	
				Led_Run:=FALSE;
				SS_MoveState:=0;
				SS_currentStep:=0;
				SS_InitStartPositionDone:=FALSE;
				//SS_StepSystemTime[SS_StepNumber]:=F_GetSysTime();
	END_CASE
END_IF
(*获取每一步耗时*)
//FOR	m:= 0 TO SS_StepNumber DO
//	SS_StepCountTime[m]:=(SS_StepSystemTime_End[m]-SS_StepSystemTime_Begin[m]);
//END_FOR

(*STOP*)
IF SS_Stop THEN
	FB_Move.BCGapReset:=TRUE;							(*¸øÔË¶¯FB¸øÍ£Ö¹ÐÅºÅ£¬Ê¹FB_Move×´Ì¬»Ö¸´*)
	FB_Move();											(*Æô¶¯FB_Move*)
	SS_Move:=FALSE;								(*btn_GapMove:=FALSE*)
	SS_MoveState:=0;										(*m_state:=0;*)
	CASE SS_StopState OF
			0:
				FB_Stop.Mode:=1;							(*1£ºgapÄ£Ê½£»2£ºµ¥ÁºÄ£Ê½£»3£ºtaperÄ£Ê½£»4£ºDebugÄ£Ê½£»5£ºBCGapÄ£Ê½*)
				FB_Stop.PowerState:=st_Power;				(*µçÔ´×´Ì¬ÊäÈë*)
				FB_Stop.BCGapStop:=TRUE;				(*Execute TRUE*)
				FB_Stop();								(*Æô¶¯FB*)
				SS_StopState:=1;
			1:
				FB_Stop();
				IF NOT FB_Stop.BCGapDone THEN			(*Í£Ö¹Î´Íê³É£¬Ñ­»·*)
					SS_StopState:=1;
				ELSE									(*Í£Ö¹Íê³É£¬ÏÂÒ»²½*)
					SS_StopState:=88;
				END_IF
			88:
				SS_Stop:=FALSE;						(*»Ö¸´×´Ì¬*)
				FB_Move.BCGapReset:=FALSE;				(*ÔËÐÐFB*)
				SS_StopState:=0;
		END_CASE
END_IF

(*触发限位开关后，相当于点击了Stop按钮*)
FTrig_ReachLS(CLK:=Unreach_LS_Far AND Unreach_LS_Near);
IF FTrig_ReachLS.Q THEN
	SS_Stop:=TRUE;
END_IF
END_ACTION

END_PROGRAM

(* stored: Version 1.1.0.1, ProductVersion 3.1.4024.6
   POU UserMode: Id {dbb58c86-3204-4c0e-a297-03b24a68bd10}, SpecialFunc None
   Action A_CheckMotorsPos: Id {f3cd81f2-82fa-493f-8c36-20c483307c7d}
   Action A_GlobalChainProtection_EPS: Id {06b22d18-fd3c-40de-ae42-96c81b461f09}
   Action A_GlobalChainProtection_MPS: Id {214f7982-b3a1-46e2-bee6-e29b232f3cd2}
   Action A_InitCompensationData: Id {1e6a9c39-c8a5-4c48-b57c-71effe5e3747}
   Action A_OneKeyToMaxGap: Id {ba9dc3e9-1e8e-4d76-8af6-498bfc77c09c}
   Action A_PowerOff: Id {e3ff8ae4-6e0c-4bb4-9a62-00e47841163f}
   Action A_PowerOn: Id {cacab3c1-f169-458e-acb8-60acf8e4d140}
   Action A_RegularMotion: Id {79d2706f-89ad-4612-adf2-c80c9fc85b18}
   Action A_SpectroscopyScanningMotion: Id {6676a965-5ff1-46e4-b651-02d2762b99bc} *)
